//==================================================================================================
//							Beckhoff Automation Poland
//									2.11.2018
//	Program inicjalizujacy prace maszyny - powinien byc wykonywany tylko w trybie E_MachineMode.eInitialization
//	Przejscie do innych trybow powinno byc mozliwe po wystawieniu flagi bInitialized
//	Program podczas inicjalizacji tlumi globalne flagi: GVL.bMuteGeneralError i GVL.bMuteGeneralFatalError
//	Reset mozliwy tylko w przypadku bledu.
//	Zawiera opsje testu - ignorujemy wowczas bledy i przechodzimy od razu do stanu bInitialized
// 	v1.0	|| TC v 3.1.4022.25		|| - Pierwsza wersja
//==================================================================================================
PROGRAM P_Initialization
VAR_INPUT
	bReset					: BOOL;
	bTestMode				: BOOL;				// Deactivate error detecton - go to initialized
END_VAR
VAR_OUTPUT
	bInitialized			: BOOL;
	bBusy					: BOOL;
	bError					: BOOL;
END_VAR
VAR
	iStep					: INT;
	rtReset					: R_TRIG;
	rtError					: R_TRIG;
	tonWatchdog				: TON;
END_VAR

// Wait some time to initialize
tonWatchdog(IN:= bBusy, PT:= T#1M, Q=> , ET=> );
rtError(CLK:= tonWatchdog.Q, Q=> );

IF rtError.Q THEN
	iStep							:= 1000;
END_IF

// Reset - reinitialize
rtReset(CLK:= bReset, Q=> );

IF bTestMode THEN
	iStep							:= 500;
END_IF

CASE iStep OF

	0: // Idle
	
		iStep	 					:= iStep + 10;
	
	10: 
	
		IF P_SystemInfo.bOK THEN
			iStep 					:= iStep + 10;
		ELSE
			// There is problem with System - usually persistent data
			P_SystemInfo.bConfirm 	:= bReset;
		END_IF
	
	20:

		IF P_EtherCAT_Diag.bOK THEN
			iStep 					:= iStep + 10;
		END_IF

	30:

		IF P_Checks.bOK THEN
			iStep 					:= iStep + 10;
		END_IF
		
	40:

		IF P_TaskInfo.bOK THEN
			iStep 					:= iStep + 10;
		END_IF
		
	50:
	// Serial No, etc
		iStep 						:= 500;
		
	500: // Initialized
	
		;
	
	1000: // Error step, wait for reset
	
		IF rtReset.Q THEN
			P_SystemInfo.bConfirm 	:= TRUE;
			iStep 					:= 0;
		END_IF;

END_CASE

bBusy 								:= iStep < 500;
bError 								:= iStep = 1000;
bInitialized						:= iStep = 500;

// Mute Errors during init phase
GVL.bMuteGeneralError				:= bBusy;
GVL.bMuteGeneralFatalError			:= bBusy;

END_PROGRAM

(* stored: Version 1.1.0.1, ProductVersion 3.1.4022.12
   POU P_Initialization: Id {97803ff5-a944-4b0c-b0e5-208abcc7a28c}, SpecialFunc None *)
